{attribute 'qualified_only'}
VAR_GLOBAL
	Case_Length_Check_Start 	: 	BOOL;
	Case_Length					:	LREAL;
	Cam_Trig					: 	BOOL;
	mastering_vision_x			:	LREAL;
	Back_Shot_Position			:	LREAL;
	Reshot_Position				:	LREAL;
	Back_Trig					: 	BOOL;
END_VAR

(* stored: Version 1.1.0.1, ProductVersion 3.1.4024.16
   GVL GVL_Mastering: Id {d0ef85e8-ecc1-44ea-9514-606fdbb4c949} *)
